FUNCTION_BLOCK _ETcVnBlobCombination_TestSuite EXTENDS TcUnit.FB_TestSuite
VAR
END_VAR

TestAddress();
TestClearReference();
TestClone();
TestTypeNameReturnsExpected();
TestIdentifierReturnsExpected();
TestMakeReferenceToFollowsReference();
TestMakeReferenceToUpdatesReference();
TestSize();
TestValueReturnsExpectedAfterInit();
TestValueReturnsExpectedAfterChange();
TestSerializeTypeWith();
TestSerializeWith();
TestTryDeserializeFrom();
TestTryMakeReferenceToFollowsReference();
TestTryMakeReferenceToUpdatesReference();

METHOD PUBLIC TestAddress
VAR
    _type : _ETcVnBlobCombination(ETcVnBlobCombination.TCVN_BC_SMALLEST);
    notExpected : PVOID := 0;
    actual : PVOID;
END_VAR
TEST('TestAddress');

actual := _type.Address;

AssertFalse(
    Condition := (notExpected = actual),
    Message := 'Type did not return a valid address.'
);

TEST_FINISHED();
END_METHOD

METHOD PUBLIC TestClearReference
VAR
    _type : _ETcVnBlobCombination(ETcVnBlobCombination.TCVN_BC_SMALLEST);
	target : ETcVnBlobCombination := ETcVnBlobCombination.TCVN_BC_SMALLEST;
    expected : ETcVnBlobCombination := ETcVnBlobCombination.TCVN_BC_SMALLEST;
    actual : ETcVnBlobCombination;
END_VAR
TEST('TestClearReference');

_type.MakeReferenceTo(target);
_type.ClearReference();
target := ETcVnBlobCombination.TCVN_BC_LARGEST;

actual := _type.Value;

AssertEquals(
    Expected := expected,
    Actual := actual,
    Message := 'Value continued to follow target.'
);

TEST_FINISHED();
END_METHOD

METHOD PUBLIC TestClone
VAR
    _type : _ETcVnBlobCombination(ETcVnBlobCombination.TCVN_BC_SMALLEST);
	clone : I_Datatype;
	isValidClone : BOOL;
	compareResult : DINT;
END_VAR
TEST('TestClone');

clone := _type.Clone();

isValidClone := clone <> 0;

IF isValidClone THEN
	compareResult := memcmp(_type.Address, clone.Address, clone.Size);
END_IF

AssertTrue(
	Condition := isValidClone,
	Message := 'Clone did not produce a clone'
);

AssertEquals_DINT(
	Expected := 0,
    Actual := compareResult,
    Message := 'Clone did not return a valid clone.'
);

clone.Dispose();

TEST_FINISHED();
END_METHOD

METHOD PUBLIC TestIdentifierReturnsExpected
VAR
    _type : _ETcVnBlobCombination(ETcVnBlobCombination.TCVN_BC_SMALLEST);
    expected : STRING := 'ETcVnBlobCombination';
    actual : STRING;
END_VAR
TEST('TestIdentifierReturnsExpected');

actual := _type.Identifier;

AssertEquals_STRING(
    Expected := expected,
    Actual := actual,
    Message := 'Type did not return correct iec type.'
);

TEST_FINISHED();
END_METHOD

METHOD PUBLIC TestMakeReferenceToFollowsReference
VAR
    _type : _ETcVnBlobCombination(ETcVnBlobCombination.TCVN_BC_SMALLEST);
	target : ETcVnBlobCombination := ETcVnBlobCombination.TCVN_BC_SMALLEST;
    expected : ETcVnBlobCombination := ETcVnBlobCombination.TCVN_BC_LARGEST;
    actual : ETcVnBlobCombination;
END_VAR
TEST('TestMakeReferenceToFollowsReference');

_type.MakeReferenceTo(target);
target := ETcVnBlobCombination.TCVN_BC_LARGEST;

actual := _type.Value;

AssertEquals(
    Expected := expected,
    Actual := actual,
    Message := 'Value did not follow target change.'
);

TEST_FINISHED();
END_METHOD

METHOD PUBLIC TestMakeReferenceToUpdatesReference
VAR
    _type : _ETcVnBlobCombination(ETcVnBlobCombination.TCVN_BC_SMALLEST);
	target : ETcVnBlobCombination := ETcVnBlobCombination.TCVN_BC_SMALLEST;
    expected : ETcVnBlobCombination := ETcVnBlobCombination.TCVN_BC_LARGEST;
    actual : ETcVnBlobCombination;
END_VAR
TEST('TestMakeReferenceToUpdatesReference');

_type.MakeReferenceTo(target);
_type.Value := ETcVnBlobCombination.TCVN_BC_LARGEST;

actual := target;

AssertEquals(
    Expected := expected,
    Actual := actual,
    Message := 'Value did not update target.'
);

TEST_FINISHED();
END_METHOD

METHOD PUBLIC TestSerializeTypeWith
VAR
    _type : _ETcVnBlobCombination(ETcVnBlobCombination.TCVN_BC_SMALLEST);
    serializer : JsonSerializer;
    expected : STRING(500) := '{"typeName":"ENUM","identifier":"ETcVnBlobCombination","enumerations":["TCVN_BC_SMALLEST","TCVN_BC_LARGEST","TCVN_BC_MIN_THRESHOLD","TCVN_BC_MAX_THRESHOLD","TCVN_BC_MEDIAN_THRESHOLD"],"baseType":{"typeName":"DINT","minValue":-2147483648,"maxValue":2147483647,"isSigned":true,"isFloat":false}}';
    actual : STRING(500);
END_VAR
TEST('TestSerializeTypeWith');

serializer.Reset();
_type.SerializeTypeWith(serializer);
serializer.TryGetSerializedData(ADR(actual), SIZEOF(actual));

AssertEquals_STRING(
    Expected := expected,
    Actual := actual,
    Message := 'Serialization of type did not return correct string.'
);

TEST_FINISHED();
END_METHOD

METHOD PUBLIC TestSerializeWith
VAR
    _type : _ETcVnBlobCombination(ETcVnBlobCombination.TCVN_BC_SMALLEST);
    serializer : JsonSerializer;
    expected : STRING := '"TCVN_BC_SMALLEST"';
    actual : STRING(500);
END_VAR
TEST('TestSerializeWith');

serializer.Reset();
_type.SerializeWith(serializer);
serializer.TryGetSerializedData(ADR(actual), SIZEOF(actual));

AssertEquals_STRING(
    Expected := expected,
    Actual := actual,
    Message := 'Serialization of type data did not return correct string.'
);

TEST_FINISHED();
END_METHOD

METHOD PUBLIC TestSize
VAR
    _type : _ETcVnBlobCombination(ETcVnBlobCombination.TCVN_BC_SMALLEST);
    expected : UDINT := SIZEOF(ETcVnBlobCombination);
    actual : UDINT;
END_VAR
TEST('TestSize');

actual := _type.Size;

AssertEquals_UDINT(
    Expected := Expected,
    Actual := actual,
    Message := 'Type did not return the correct size.'
);

TEST_FINISHED();
END_METHOD

METHOD PUBLIC TestTryDeserializeFrom
VAR
    deserializer : JsonDeserializer;
    feedback : DeserializerFeedback;
    json : STRING := '"TCVN_BC_SMALLEST"';
    _type : _ETcVnBlobCombination(ETcVnBlobCombination.TCVN_BC_SMALLEST);
    expected : ETcVnBlobCombination := ETcVnBlobCombination.TCVN_BC_SMALLEST;
    actual : ETcVnBlobCombination;
 END_VAR
TEST('TestTryDeserializeFrom');

deserializer.Reset();
deserializer.TryLoad(json);
_type.TryDeserializeFrom(Deserializer, Feedback);

actual := _type.Value;

AssertEquals(
    Expected := expected,
    Actual := actual,
    Message := 'Type did not deserialize correctly.'
);

TEST_FINISHED();
END_METHOD

METHOD PUBLIC TestTryMakeReferenceToFollowsReference
VAR
    _type : _ETcVnBlobCombination(ETcVnBlobCombination.TCVN_BC_SMALLEST);
	target : _ETcVnBlobCombination(ETcVnBlobCombination.TCVN_BC_SMALLEST);
    expected : ETcVnBlobCombination := ETcVnBlobCombination.TCVN_BC_LARGEST;
    actual : ETcVnBlobCombination;
END_VAR
TEST('TestTryMakeReferenceToFollowsReference');

_type.TryMakeReferenceTo(target);
target.Value := ETcVnBlobCombination.TCVN_BC_LARGEST;

actual := _type.Value;

AssertEquals(
    Expected := expected,
    Actual := actual,
    Message := 'Value did not follow target change.'
);

TEST_FINISHED();
END_METHOD

METHOD PUBLIC TestTryMakeReferenceToUpdatesReference
VAR
    _type : _ETcVnBlobCombination(ETcVnBlobCombination.TCVN_BC_SMALLEST);
	target : _ETcVnBlobCombination(ETcVnBlobCombination.TCVN_BC_SMALLEST);
    expected : ETcVnBlobCombination := ETcVnBlobCombination.TCVN_BC_LARGEST;
    actual : ETcVnBlobCombination;
END_VAR
TEST('TestTryMakeReferenceToUpdatesReference');

_type.TryMakeReferenceTo(target);
_type.Value := ETcVnBlobCombination.TCVN_BC_LARGEST;

actual := target.Value;

AssertEquals(
    Expected := expected,
    Actual := actual,
    Message := 'Value did not update target.'
);

TEST_FINISHED();
END_METHOD

METHOD PUBLIC TestTypeNameReturnsExpected
VAR
    _type : _ETcVnBlobCombination(ETcVnBlobCombination.TCVN_BC_SMALLEST);
    expected : STRING := 'ENUM';
    actual : STRING;
END_VAR
TEST('TestTypeNameReturnsExpected');

actual := _type.TypeName;

AssertEquals_STRING(
    Expected := expected,
    Actual := actual,
    Message := 'Type did not return correct iec type.'
);

TEST_FINISHED();
END_METHOD

METHOD PUBLIC TestValueReturnsExpectedAfterChange
VAR
    _type : _ETcVnBlobCombination(ETcVnBlobCombination.TCVN_BC_SMALLEST);
    expected : ETcVnBlobCombination := ETcVnBlobCombination.TCVN_BC_LARGEST;
    actual : ETcVnBlobCombination;
END_VAR
TEST('TestValueReturnsExpectedAfterChange');

_type.Value := ETcVnBlobCombination.TCVN_BC_LARGEST;

actual := _type.Value;

AssertEquals(
    Expected := expected,
    Actual := actual,
    Message := 'Expected value not returned after change.'
);

TEST_FINISHED();
END_METHOD

METHOD PUBLIC TestValueReturnsExpectedAfterInit
VAR
    _type : _ETcVnBlobCombination(ETcVnBlobCombination.TCVN_BC_SMALLEST);
    expected : ETcVnBlobCombination := ETcVnBlobCombination.TCVN_BC_SMALLEST;
    actual : ETcVnBlobCombination;
END_VAR
TEST('TestValueReturnsExpectedAfterInit');

actual := _type.Value;

AssertEquals(
    Expected := expected,
    Actual := actual,
    Message := 'Expected value not returned after Init.'
);

TEST_FINISHED();
END_METHOD

END_FUNCTION_BLOCK

(* stored: Version 1.1.0.1, ProductVersion 3.1.4024.12
   POU _ETcVnBlobCombination_TestSuite: Id {643d61d1-ad26-0df9-2d62-f145356bf4b8}, SpecialFunc None
   Method TestAddress: Id {772c8f8f-3479-0060-0fd2-487c46470f2e}
   Method TestClearReference: Id {f98a377c-fe88-0873-2a4e-4222f19c580b}
   Method TestClone: Id {45d8f60a-5fe7-07ea-23cf-e217f1e7ecab}
   Method TestIdentifierReturnsExpected: Id {37dfcf7f-e677-0fb0-3a99-3b9f55364738}
   Method TestMakeReferenceToFollowsReference: Id {7d7e7d0f-07c8-0e2a-22e6-356b36fb6cfe}
   Method TestMakeReferenceToUpdatesReference: Id {290eb901-f7c5-0e86-3ef5-44b5d43d82c6}
   Method TestSerializeTypeWith: Id {428dd906-7041-0b44-2143-84b984aa782c}
   Method TestSerializeWith: Id {9c0eccff-c772-0d1e-2464-94585b3e8f85}
   Method TestSize: Id {a106d3c5-0d8d-0fc0-3961-6086bcf868b7}
   Method TestTryDeserializeFrom: Id {951a5151-ed4f-00e0-350b-cf07237a11dc}
   Method TestTryMakeReferenceToFollowsReference: Id {f83ba383-b38e-0c31-3438-c68578e261a1}
   Method TestTryMakeReferenceToUpdatesReference: Id {6374d5cd-8422-07b0-39b9-a82be7742846}
   Method TestTypeNameReturnsExpected: Id {43c5ba03-0125-0ded-0175-d08ff3c41e17}
   Method TestValueReturnsExpectedAfterChange: Id {d1a1aa89-085d-077b-19e2-aea000b5467b}
   Method TestValueReturnsExpectedAfterInit: Id {b465ceea-209a-0c7b-39de-d77232ddc53f} *)
